{attribute 'qualified_only'}
VAR_GLOBAL
	GrindingWheelMS AT %Q* : BOOL;
	StartGrindingWheelPB AT %I* : BOOL;
	StopGrindingWheelPB AT %I*  : BOOL;
END_VAR

(* stored: Version 1.1.0.1, ProductVersion 3.1.4024.4
   GVL Grinder: Id {e568357a-3c8c-494a-bbc5-d71ff6895687} *)
